FUNCTION testReferenceToFB :ARRAY [1..2]OF  REAL
VAR_INPUT
	RefSum: REFERENCE TO mySumFb;
	PointerSum: POINTER TO mySumFb;
	sum2:REAL;
END_VAR
VAR
		MyFb_p_Sum:mySumFb;
END_VAR

MyFb_p_Sum := PointerSum^;

RefSum.sum2:=sum2;
testReferenceToFB[1]:=MyFb_p_Sum.result;
testReferenceToFB[2]:=RefSum.result;

END_FUNCTION

(* stored: Version 1.1.0.1, ProductVersion 3.1.4024.6
   POU testReferenceToFB: Id {eaa6da5b-ba98-4b45-b796-0484949e48c4}, SpecialFunc None *)
